FUNCTION_BLOCK Seq_Set_Plate_1 EXTENDS FB_BASIS IMPLEMENTS I_Sequenz
VAR_INPUT
	// Benötigte Skills
	Move_Robot			:I_Skill_Roboter;
	
	// Benötigte Parameter
	R_Plate_Pos			:sRoboterProzessVariablen; 
	R_Offset_X			:LREAL;
	R_Offset_Y			:LREAL;
	R_Offset_Z			:LREAL;
	
END_VAR
VAR_OUTPUT
END_VAR
VAR
	R_Offset_X_Pos		:sRoboterProzessVariablen; 
	R_Offset_Y_Pos		:sRoboterProzessVariablen; 
	R_Offset_Z_Pos		:sRoboterProzessVariablen; 
END_VAR

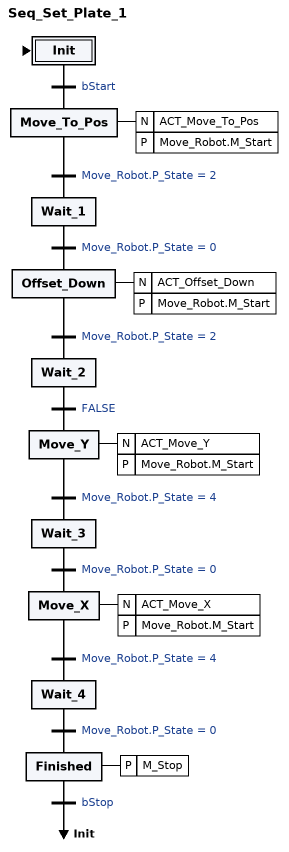
INITIAL_STEP Init:
END_STEP
TRANSITION FROM Init TO Move_To_Pos
    := bStart;
END_TRANSITION
STEP Move_To_Pos:
    ACT_Move_To_Pos(N);
    Move_Robot.M_Start(P);
END_STEP
TRANSITION FROM Move_To_Pos TO Wait_1
    := Move_Robot.P_State = 2;
END_TRANSITION
STEP Wait_1:
END_STEP
TRANSITION FROM Wait_1 TO Offset_Down
    := Move_Robot.P_State = 0;
END_TRANSITION
STEP Offset_Down:
    ACT_Offset_Down(N);
    Move_Robot.M_Start(P);
END_STEP
TRANSITION FROM Offset_Down TO Wait_2
    := Move_Robot.P_State = 2;
END_TRANSITION
STEP Wait_2:
END_STEP
TRANSITION FROM Wait_2 TO Move_Y
    := FALSE;
END_TRANSITION
STEP Move_Y:
    ACT_Move_Y(N);
    Move_Robot.M_Start(P);
END_STEP
TRANSITION FROM Move_Y TO Wait_3
    := Move_Robot.P_State = 4;
END_TRANSITION
STEP Wait_3:
END_STEP
TRANSITION FROM Wait_3 TO Move_X
    := Move_Robot.P_State = 0;
END_TRANSITION
STEP Move_X:
    ACT_Move_X(N);
    Move_Robot.M_Start(P);
END_STEP
TRANSITION FROM Move_X TO Wait_4
    := Move_Robot.P_State = 4;
END_TRANSITION
STEP Wait_4:
END_STEP
TRANSITION FROM Wait_4 TO Finished
    := Move_Robot.P_State = 0;
END_TRANSITION
STEP Finished:
    M_Stop(P);
END_STEP
TRANSITION FROM Finished TO Init
    := bStop;
END_TRANSITION

ACTION ACT_Move_To_Pos:
Move_Robot.P_Prozessparameter := R_Plate_Pos;
END_ACTION

ACTION ACT_Move_X:
R_Offset_X_Pos.q1 := -R_Offset_X;
R_Offset_X_Pos.v := 0.1;
R_Offset_X_Pos.a := 0.1;
R_Offset_X_Pos.MoveTyp := 0;
R_Offset_X_Pos.PosTyp := 1;

Move_Robot.P_Prozessparameter := R_Offset_X_Pos;
END_ACTION

ACTION ACT_Move_Y:
R_Offset_Y_Pos.q1 := -R_Offset_Y;
R_Offset_Y_Pos.v := 0.1;
R_Offset_Y_Pos.a := 0.1;
R_Offset_Y_Pos.MoveTyp := 0;
R_Offset_Y_Pos.PosTyp := 1;

Move_Robot.P_Prozessparameter := R_Offset_Y_Pos;
END_ACTION

ACTION ACT_Offset_Down:
R_Offset_Z_Pos.q3 := -R_Offset_Z;
R_Offset_Z_Pos.v := 0.1;
R_Offset_Z_Pos.a := 0.1;
R_Offset_Z_Pos.MoveTyp := 0;
R_Offset_Z_Pos.PosTyp := 1;

Move_Robot.P_Prozessparameter := R_Offset_Z_Pos;
END_ACTION

END_FUNCTION_BLOCK

(* stored: Version 1.1.0.1
   POU Seq_Set_Plate_1: Id {e4fbf3e6-48ad-45ed-83d4-04f0824110a3}, SpecialFunc None
   Folder 01_Zuwesiung: Id {ff494c44-2a08-4e42-87ce-ff58bd56d01e}
   Action ACT_Move_To_Pos: Id {3398db22-565c-4628-8f96-bc8238b0d037}
   Action ACT_Move_X: Id {a53982f1-8bc8-4739-888e-bfed478ade3e}
   Action ACT_Move_Y: Id {d81287df-a8c3-4c46-839c-69e65da09ad6}
   Action ACT_Offset_Down: Id {2c2e691b-7708-4eba-97ea-4e1451519df5} *)
